FUNCTION_BLOCK FB_CleaningProcessStateService EXTENDS FB_CleaningProcessStateBase
VAR_INPUT
END_VAR
VAR_OUTPUT
END_VAR
VAR

END_VAR

METHOD mCleaningOp : BOOL
VAR_INPUT
	sI_Operation : EN_CLEANING_OP;
END_VAR
//Switch to production mode if no operation active
IF I_MachineStatus.pSafetyOk AND I_MachineStatus.pMachineReady AND NOT bL_DevOpActive THEN
  IF sI_Operation = eOPCAPENTER THEN
    I_ParentCallback.mChangeState(EN_Cleaning_State.Capping);
  ELSIF sI_Operation = eOPCAPEXIT THEN
    I_ParentCallback.mChangeState(EN_Cleaning_State.CappingExit);
  ELSIF sI_Operation = eOPCLEAN THEN
    I_ParentCallback.mChangeState(EN_Cleaning_State.Cleaning);
  ELSIF sI_Operation = eOPPURGE THEN
    I_ParentCallback.mChangeState(EN_Cleaning_State.Capping);
  END_IF
END_IF
END_METHOD

METHOD mEntryAction
VAR_INPUT
END_VAR
iL_CurrentStep := 0;

// Launch initial command to bring system to service mode
bL_DevOpActive := I_ParentCallback.mSetMode(EN_CLEANING_OP.eOPPREPSERVICE);
END_METHOD

METHOD mProduction : BOOL
VAR_INPUT
END_VAR
//Switch to production mode if no operation active
IF I_MachineStatus.pSafetyOk AND I_MachineStatus.pMachineReady AND NOT bL_DevOpActive THEN
	I_ParentCallback.mChangeState(EN_Cleaning_State.Production);
END_IF
END_METHOD

METHOD mService : BOOL
VAR_INPUT
END_VAR
//Request service mode - implement in SubClass
mService := TRUE;
END_METHOD

METHOD mStateAction
VAR_INPUT
END_VAR

VAR
	sL_DeviceStatus: ST_CLEANING_DEV_STATUS;
END_VAR
sL_DeviceStatus := I_ParentCallback.pDeviceStatus;

IF bL_DevOpActive THEN
	mDevOp();
END_IF

//If error go to error mode
IF sL_DeviceStatus.bError THEN
	I_ParentCallback.mChangeState(EN_Cleaning_State.Error);
END_IF

SUPER^.pInitDone := TRUE;
END_METHOD

END_FUNCTION_BLOCK

(* stored: Version 1.1.0.1, ProductVersion 3.1.4024.11
   POU FB_CleaningProcessStateService: Id {f161f18f-ce22-46b1-89bb-5fb825c88fd5}, SpecialFunc None
   Method mCleaningOp: Id {265d2af1-1567-4a03-8d71-f8ddf131a9da}
   Method mEntryAction: Id {f5c06c97-7d74-47e7-a6f2-14abd905009e}
   Method mProduction: Id {08cb4085-fb61-4152-a337-485e6ec842f1}
   Method mService: Id {79305885-ba2e-4106-942a-baddb62d084c}
   Method mStateAction: Id {6653e122-5fa0-49a0-b970-3a08c73622d9} *)
